// TwinCAT 3 PLC project Untitled2
// ProgramVersion: 3.1.4023.0
// libraries:
//   Tc2_Standard, * (Beckhoff Automation GmbH)
//   Tc2_System, * (Beckhoff Automation GmbH)
//   Tc3_Module, * (Beckhoff Automation GmbH)
// project tree:
//   GVLs/ GVL.TcGVL
//   / PlcTask.TcTTO
//   POUs/ MAIN.TcPOU
// real-time tasks:
//   TASK PlcTask: cycle T#10ms, priority 20, ADS port 350
// I/O:
//   DEVICE Device 1 (EtherCAT), AmsNetId 192.168.56.1.2.1
//     Term 1 (EK1101) [EK1101 EtherCAT Coupler (2A E-Bus, ID switch)]
//       Term 2 (EL6910) [EL6910, TwinSAFE PLC]
//       Term 3 (EL1904) [EL1904, 4 Ch. Safety Input 24V, TwinSAFE]
//         modules: Module 1 (FSOES)
//       Term 4 (EL2904) [EL2904, 4 Ch. Safety Output 24V, 0.5A, TwinSAFE]
//         modules: Module 1 (FSOES), Module 2 (DO)
// variable links:
//   (this object) <-> Device 1 (EtherCAT)/Term 1 (EK1101)/Term 2 (EL6910)
//     Term 1 (EK1101)/Term 3 (EL1904)/Module 1 (FSOES)/RxPDO/FSOE <-> ConnectionInputs/Message_2 TxPDO
//     Term 1 (EK1101)/Term 3 (EL1904)/Module 1 (FSOES)/TxPDO/FSOE <-> ConnectionOutputs/Message_2 RxPDO
//   (this object) <-> Device 1 (EtherCAT)/Term 1 (EK1101)/Term 3 (EL1904)
//     Term 1 (EK1101)/Term 2 (EL6910)/ConnectionInputs/Message_2 TxPDO <-> Module 1 (FSOES)/RxPDO/FSOE
//     Term 1 (EK1101)/Term 2 (EL6910)/ConnectionOutputs/Message_2 RxPDO <-> Module 1 (FSOES)/TxPDO/FSOE
//   Untitled2 Instance <-> Device 1 (EtherCAT)/Term 1 (EK1101)/Term 2 (EL6910)
//     PlcTask Inputs/GVL.SafetyAndOut <-> StandardInputs/TwinSafeGroup1.Std_OutSafety_4
//     PlcTask Outputs/GVL.ErrAck <-> StandardOutputs/TwinSafeGroup1.ErrorAcknowledgement_1
//     PlcTask Outputs/GVL.RunStop <-> StandardOutputs/TwinSafeGroup1.Std_RunStop_3

CONFIGURATION Untitled2
    RESOURCE PLC ON TwinCAT3
        TASK PlcTask(INTERVAL := T#10ms, PRIORITY := 20);
        PROGRAM MAIN WITH PlcTask : MAIN;
    END_RESOURCE
END_CONFIGURATION

// ---- GVLs/GVL.TcGVL
{attribute 'qualified_only'}
VAR_GLOBAL
	RunStop			AT %Q*	: BOOL;
	ErrAck			AT %Q*	: BOOL;
	
	SafetyAndOut	AT %I*	: BOOL;
	
END_VAR

// ---- POUs/MAIN.TcPOU
PROGRAM MAIN
VAR
END_VAR

END_PROGRAM
